{region '#Template'}
	{attribute 'Version' := '1.0.0.0'}
	{attribute 'Tags' := '"LCID": "1031", "Text": "AC, Setpoint, Room temperature"'}
	{attribute 'Tags' := '"LCID": "1033", "Text": "AC, Setpoint, Room temperature"'}
	{attribute 'Description' := '"LCID": "1031", "Text": "Sollwert Raumtemperatur"'}
	{attribute 'Description' := '"LCID": "1033", "Text": "Setpoint room temperature"'}
{endregion}
FUNCTION_BLOCK FB_BA_AC_SpTRm_01 EXTENDS FB_BA_View
VAR_INPUT
	fTWth					: REAL;	
END_VAR
VAR_OUTPUT
	fSp						: REAL;
END_VAR
VAR_INPUT CONSTANT
	X1						: FB_BA_AV_Op;
	X2						: FB_BA_AV_Op;
	X3						: FB_BA_AV_Op;
	X4						: FB_BA_AV_Op;
	Y1						: FB_BA_AV_Op;
	Y2_3					: FB_BA_AV_Op;	
	Y4						: FB_BA_AV_Op;
	Sp						: FB_BA_AV_Op;						
END_VAR
VAR
	Scale					: FB_BA_Chrct04;	
END_VAR

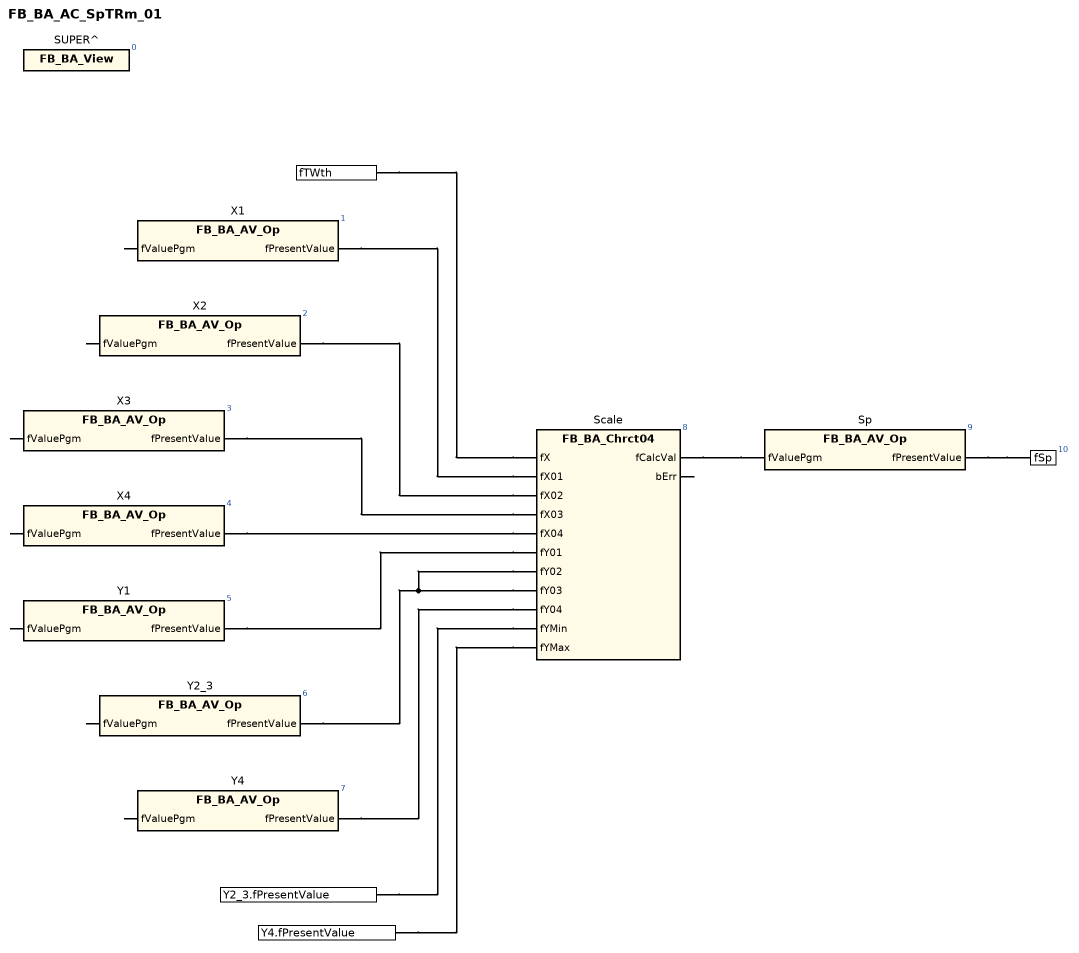
SUPER^(); // FB_BA_View
X1(); // FB_BA_AV_Op
X2(); // FB_BA_AV_Op
X3(); // FB_BA_AV_Op
X4(); // FB_BA_AV_Op
Y1(); // FB_BA_AV_Op
Y2_3(); // FB_BA_AV_Op
Y4(); // FB_BA_AV_Op
Scale(
    fX := fTWth,
    fX01 := X1.fPresentValue,
    fX02 := X2.fPresentValue,
    fX03 := X3.fPresentValue,
    fX04 := X4.fPresentValue,
    fY01 := Y1.fPresentValue,
    fY02 := Y2_3.fPresentValue,
    fY03 := Y2_3.fPresentValue,
    fY04 := Y4.fPresentValue,
    fYMin := Y2_3.fPresentValue,
    fYMax := Y4.fPresentValue); // FB_BA_Chrct04
Sp(fValuePgm := Scale.fCalcVal); // FB_BA_AV_Op
fSp := Sp.fPresentValue;

METHOD FB_init : BOOL
VAR_INPUT
	bInitRetains : BOOL; // if TRUE, the retain variables are initialized (warm start / cold start)
	bInCopyCode : BOOL;  // if TRUE, the instance afterwards gets moved into the copy code (online change)
END_VAR
X1.iParent				:= THIS^;
X1.iLabel				:= LblCmpAC.SpTRm_X1;			
X1.sObjectName			:= '{Idx=01}';								 	 
X1.eUnit				:= E_BA_Unit.eTemperature_DegreesCelsius;  
X1.fValueRm				:= -15.0;
X1.fCOVIncrement		:= BA2_Param.fDefCOVIncrement;

X2.iParent				:= THIS^;
X2.iLabel				:= LblCmpAC.SpTRm_X2;			
X2.sObjectName			:= '{Idx=02}';	 	 
X2.eUnit				:= E_BA_Unit.eTemperature_DegreesCelsius;  
X2.fValueRm				:= -5.0;
X2.fCOVIncrement		:= BA2_Param.fDefCOVIncrement;

X3.iParent				:= THIS^;
X3.iLabel				:= LblCmpAC.SpTRm_X3;			
X3.sObjectName			:= '{Idx=03}';								 	 
X3.eUnit				:= E_BA_Unit.eTemperature_DegreesCelsius;  
X3.fValueRm				:= 26.0;
X3.fCOVIncrement		:= BA2_Param.fDefCOVIncrement;

X4.iParent				:= THIS^;
X4.iLabel				:= LblCmpAC.SpTRm_X4;			
X4.sObjectName			:= '{Idx=04}';								 	 
X4.eUnit				:= E_BA_Unit.eTemperature_DegreesCelsius;  
X4.fValueRm				:= 32.0;
X4.fCOVIncrement		:= BA2_Param.fDefCOVIncrement;

Y1.iParent				:= THIS^;
Y1.iLabel				:= LblCmpAC.SpTRm_Y1;			
Y1.sObjectName			:= '{Idx=01}';								 	 
Y1.eUnit				:= E_BA_Unit.eTemperature_DegreesCelsius;  
Y1.fValueRm				:= 23.0;
Y1.fCOVIncrement		:= BA2_Param.fDefCOVIncrement;

Y2_3.iParent			:= THIS^;
Y2_3.iLabel				:= LblCmpAC.SpTRm_Y2_3;			
Y2_3.sObjectName		:= '{Idx=02}';								 	 
Y2_3.eUnit				:= E_BA_Unit.eTemperature_DegreesCelsius;  
Y2_3.fValueRm			:= 21.0;
Y2_3.fCOVIncrement		:= BA2_Param.fDefCOVIncrement;
	
Y4.iParent				:= THIS^;
Y4.iLabel				:= LblCmpAC.SpTRm_Y4;			
Y4.sObjectName			:= '{Idx=04}';								 	 
Y4.eUnit				:= E_BA_Unit.eTemperature_DegreesCelsius;  
Y4.fValueRm				:= 28.0;
Y4.fCOVIncrement		:= BA2_Param.fDefCOVIncrement;

Sp.iParent				:= THIS^;
Sp.iLabel				:= LblCmpAC.SpTRm_Sp;			
Sp.sObjectName			:= '{Idx=01}';								 	 
Sp.eUnit				:= E_BA_Unit.eTemperature_DegreesCelsius;
Sp.fCOVIncrement		:= BA2_Param.fDefCOVIncrement;
END_METHOD

END_FUNCTION_BLOCK

(* stored: Version 1.1.0.1, ProductVersion 3.1.4024.9
   POU FB_BA_AC_SpTRm_01: Id {c57dab52-c056-4cc8-944a-6c47ad70f6b1}, SpecialFunc None
   Method FB_init: Id {b9b66a78-c1e3-455f-99ca-e5511b0116ee} *)
